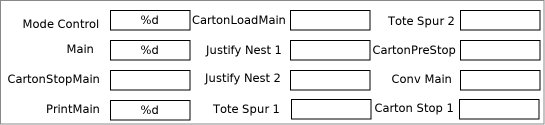
VISUALIZATION StateDisplay  // 545x125
    Rectangle (2,9 100x30), "Mode Control"
    Rectangle (110,10 80x20), "%d", text variable: Stn053_00_ModeControl.Local.State
    Rectangle (17,34 80x30), "Main"
    Rectangle (110,40 80x20), "%d", text variable: Stn053_05_StnMain.Local.State
    Rectangle (184,68 100x20), "Justify Nest 2"
    Rectangle (290,70 80x20)
    Rectangle (355,69 100x20), "Conv Main"
    Rectangle (460,70 80x20)
    Rectangle (3,69 100x20), "CartonStopMain"
    Rectangle (110,70 80x20)
    Rectangle (189,10 100x20), "CartonLoadMain"
    Rectangle (290,10 80x20)
    Rectangle (358,11 100x20), "Tote Spur 2"
    Rectangle (460,10 80x20)
    Rectangle (359,40 100x20), "CartonPreStop"
    Rectangle (460,40 80x20)
    Rectangle (185,40 100x20), "Justify Nest 1"
    Rectangle (290,40 80x20)
    Rectangle (183,99 100x20), "Tote Spur 1"
    Rectangle (291,99 80x20)
    Rectangle (17,99 86x20), "PrintMain"
    Rectangle (110,100 80x20), "%d"
    Rectangle (371,98 86x20), "Carton Stop 1"
    Rectangle (459,99 80x20)
    Rectangle (533,70 100x20), "CartonNest2"
    Rectangle (638,71 80x20)
    Rectangle (536,12 100x20), "Carton Stop 2"
    Rectangle (638,11 80x20)
    Rectangle (533,41 100x20), "CartonNest1"
    Rectangle (638,41 80x20)
    Rectangle (549,99 86x20), "Cling 1"
    Rectangle (637,100 80x20)
END_VISUALIZATION

(* stored: Version 1.1.0.1, ProductVersion 3.1.4024.6
   Visu StateDisplay: Id {f0f02838-db08-4a5c-bea6-d62f4eac4088} *)
